PROGRAM MAIN
VAR
	suctionLeft : PneumaticUnit;
	suctionRight : PneumaticUnit;
	
	enableL : BOOL;
	enableR : BOOL;
END_VAR

suctionLeft.enable := enableL;
suctionRight.enable := enableR;

END_PROGRAM

(* stored: Version 1.1.0.1, ProductVersion 3.1.4024.11
   POU MAIN: Id {98b5f675-dd89-4510-87f3-6dab8b969718}, SpecialFunc None *)
